TYPE (* IEC61131-3, Table 14#5 *)
  (* Standard: 1131-3 *)
  (* Version 0.0, 3/17/2026, Schneider Electric, Template *)
  PACKAGE Main;
  {SET_ATTRIBUTE(nxtDataType, yuBjJmbjdzTXbTqqCuFqq4iYuyX+NOw87GLmAa8/l8g8S0GssKRBD3Bw9f3nDpbvm/lpTqhTEUa7h4d7KB7HGe8iQDf7yE6aU188Q1/TVhKl8+8xnXK+A1Gzs3cfU4syGh48GTVWHsCI3HnBvYCa8yQnZNo6nXFNfvVO9q9Uz0xt2qaQzFox1tkW5mKg51wG+x+WakaohzrGwsveTM0g1psCjHlv+ekPCoDSQwJPo7KlFYNstsj5F2FtN0SahTUX81uYuRtqfwVFIWq4PrfUTsuTILCnV4iGurFOCxoDAQRkMgNFBFqYFGnyS9mqYb002CCh6sUF63elLwNKbAgS+wEnLiu2yrMJnV5rx+f7INPAPJ1J4LyewihwDwaFV/TsCJ+jJvGYYOQnaqp9wT+6ecl2ztmR0j2S)}
  Component_State_Msg : STRUCT
    src_id : INT;
    source_name : STRING[150];
    dest_name : STRING[150];
    state : INT;
  END_STRUCT;
END_TYPE
